FUNCTION_BLOCK analog_scaling
VAR_INPUT
	//Raw Input value
	raw_input : REAL;
	//Raw Input Minimum Scaling Value
	raw_min : REAL :=0;
	//Raw Input Maximum Scaling Value
	raw_max : REAL :=32767;
	//Engineering Units Minimum Scaling Value
	eu_min : REAL;
	//Engineering Units Maximum Scaling Value
	eu_max : REAL;
	//Averaging Filter Time Setpoint
	filter_factor : REAL;
END_VAR
VAR_OUTPUT
	//Scaled Value for Output
	scaled_value : REAL;
END_VAR
VAR
	//Scratchpad Value
	normalized_value : REAL;
	//unfiltered Scaled Value
	unfiltered_value : REAL;
END_VAR

//Initialize Raw_Max and EU_Max to avoid Scaled_Value=Not a number
IF raw_max = 0 AND raw_min = 0 THEN
	raw_max:=1;
END_IF
IF eu_max = 0 AND eu_min = 0 THEN
	eu_max:=1;
END_IF

//Normalize the Analog Input
IF raw_input < raw_min THEN
		normalized_value := raw_min;
	ELSIF raw_input > raw_max THEN
		normalized_value := raw_max;
	ELSE
		normalized_value := (raw_input - raw_min) / (raw_max - raw_min);
	END_IF
	
//Scale the Output
unfiltered_value := normalized_value * (eu_max-eu_min)+eu_min;

//Low Pass Filter for the output.  Increase Filter to dampen reading
scaled_value := ((scaled_value * filter_factor) + unfiltered_value) / (filter_factor +1);

END_FUNCTION_BLOCK

(* stored: Version 1.1.0.1, ProductVersion 3.1.4024.12
   POU analog_scaling: Id {6e091dc3-dcd3-4ed3-97fe-a4b8777a6a5d}, SpecialFunc None *)
